# EPICS autosave request: utcaApp/Db/fofb_processing_channel.req
$(S)$(RTM_CHAN)FOFBAccDecimation-SP
$(S)$(RTM_CHAN)FOFBAccFreeze-Sel
$(S)$(RTM_CHAN)FOFBAccSatMax-SP
$(S)$(RTM_CHAN)FOFBAccSatMin-SP
$(S)$(RTM_CHAN)InvRespMatRowX-SP
$(S)$(RTM_CHAN)InvRespMatRowY-SP
$(S)$(RTM_CHAN)FOFBAccFilter-SP
$(S)$(RTM_CHAN)FOFBAccFilterGain-SP
